// TIA Portal V17 export
// export: Created 2024-08-29T18:23:44.282771Z, ExportSetting WithDefaults, DisplayName Totally Integrated Automation Portal, DisplayVersion V17 Update 7, DisplayName TIA Portal Openness, DisplayVersion V17 Update 7, DisplayName TIA Portal Version Control Interface, DisplayVersion V17, DisplayName SINAMICS Startdrive Advanced, DisplayVersion V17 SP2, DisplayName SINAMICS Startdrive G110M, G120, G120C, G120D, G120P, G115D, DisplayVersion V17 SP2, DisplayName SINAMICS Startdrive G130, G150, S120, S150, SINAMICS MV, S210, DisplayVersion V17 SP2, DisplayName STEP 7 Professional, DisplayVersion V17 Update 7, DisplayName STEP 7 Safety, DisplayVersion V17 Update 6, DisplayName WinCC Advanced / Unified PC, DisplayVersion V17 Update 7
FUNCTION "modifyRecipe" : Void   // FC6, LAD
{ S7_Optimized_Access := 'TRUE' }
VERSION : 0.1
// stored: AutoNumber true, IsIECCheckEnabled false, SetENOAutomatically false, UDAEnableTagReadback false
   VAR_TEMP   // added for the SCL form of the ladder/FBD networks
      _w1 : Bool;
      _w2 : Bool;
   END_VAR
BEGIN

REGION Network 1: ERASE A STEP
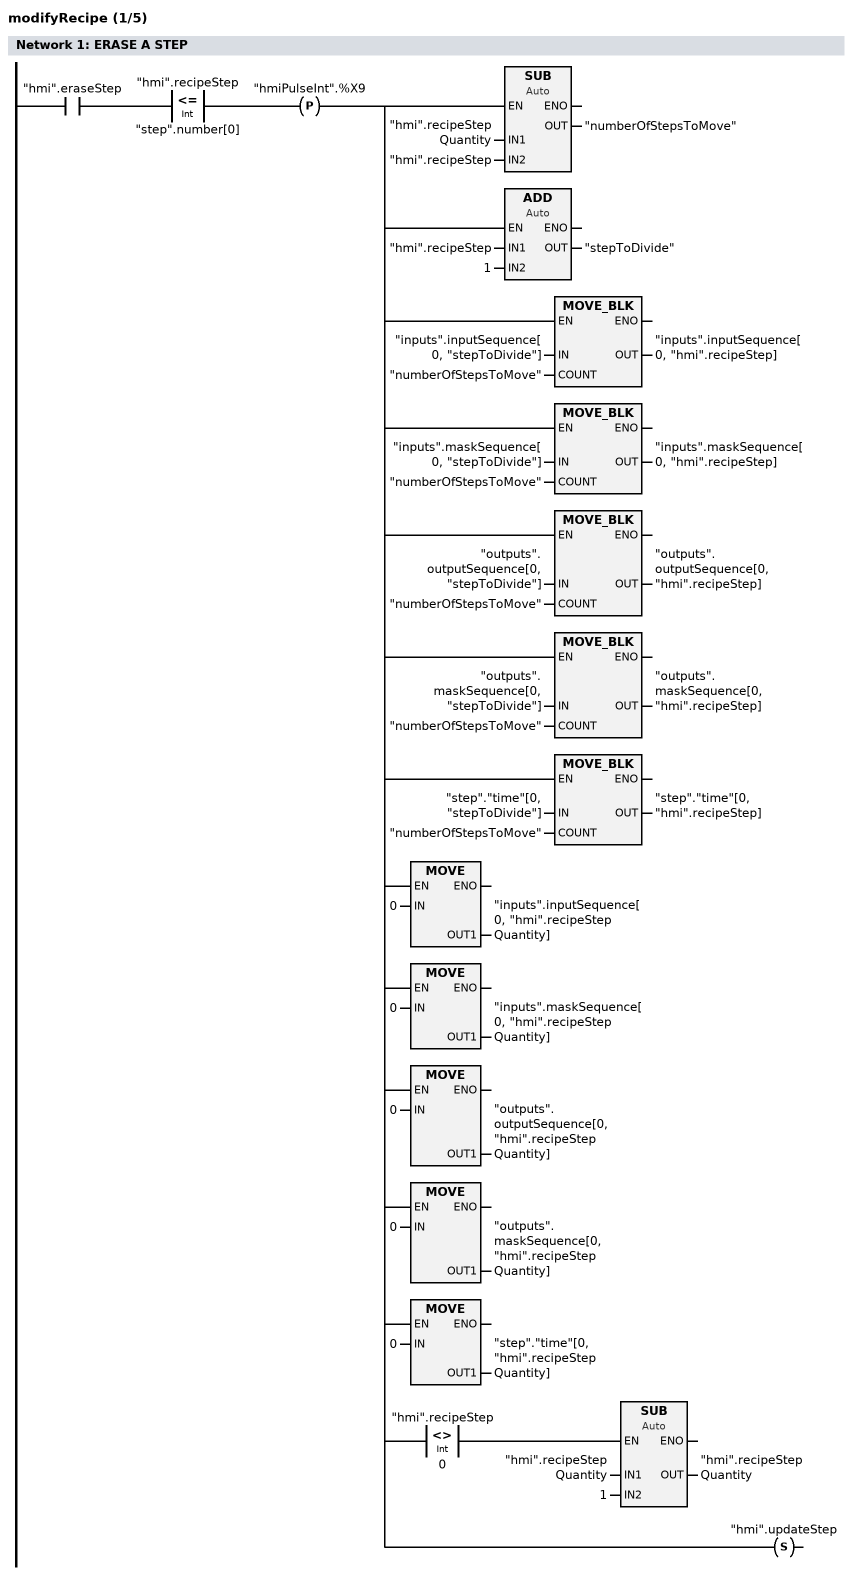
   #_w1 := "hmi".eraseStep AND ("hmi".recipeStep <= "step".number[0]);
   #_w2 := #_w1 AND NOT "hmiPulseInt".%X9;   // rising edge
   "hmiPulseInt".%X9 := #_w1;
   IF #_w2 THEN
       "numberOfStepsToMove" := "hmi".recipeStepQuantity - "hmi".recipeStep;
       "stepToDivide" := "hmi".recipeStep + 1;
       MOVE_BLK(IN := "inputs".inputSequence[0, "stepToDivide"],
                COUNT := "numberOfStepsToMove",
                OUT => "inputs".inputSequence[0, "hmi".recipeStep]);
       MOVE_BLK(IN := "inputs".maskSequence[0, "stepToDivide"],
                COUNT := "numberOfStepsToMove",
                OUT => "inputs".maskSequence[0, "hmi".recipeStep]);
       MOVE_BLK(IN := "outputs".outputSequence[0, "stepToDivide"],
                COUNT := "numberOfStepsToMove",
                OUT => "outputs".outputSequence[0, "hmi".recipeStep]);
       MOVE_BLK(IN := "outputs".maskSequence[0, "stepToDivide"],
                COUNT := "numberOfStepsToMove",
                OUT => "outputs".maskSequence[0, "hmi".recipeStep]);
       MOVE_BLK(IN := "step"."time"[0, "stepToDivide"],
                COUNT := "numberOfStepsToMove",
                OUT => "step"."time"[0, "hmi".recipeStep]);
       "inputs".inputSequence[0, "hmi".recipeStepQuantity] := 0;
       "inputs".maskSequence[0, "hmi".recipeStepQuantity] := 0;
       "outputs".outputSequence[0, "hmi".recipeStepQuantity] := 0;
       "outputs".maskSequence[0, "hmi".recipeStepQuantity] := 0;
       "step"."time"[0, "hmi".recipeStepQuantity] := 0;
   END_IF;
   IF #_w2 AND ("hmi".recipeStep <> 0) THEN "hmi".recipeStepQuantity := "hmi".recipeStepQuantity - 1; END_IF;
   IF #_w2 THEN "hmi".updateStep := TRUE; END_IF;
END_REGION

REGION Network 2: ADD A STEP
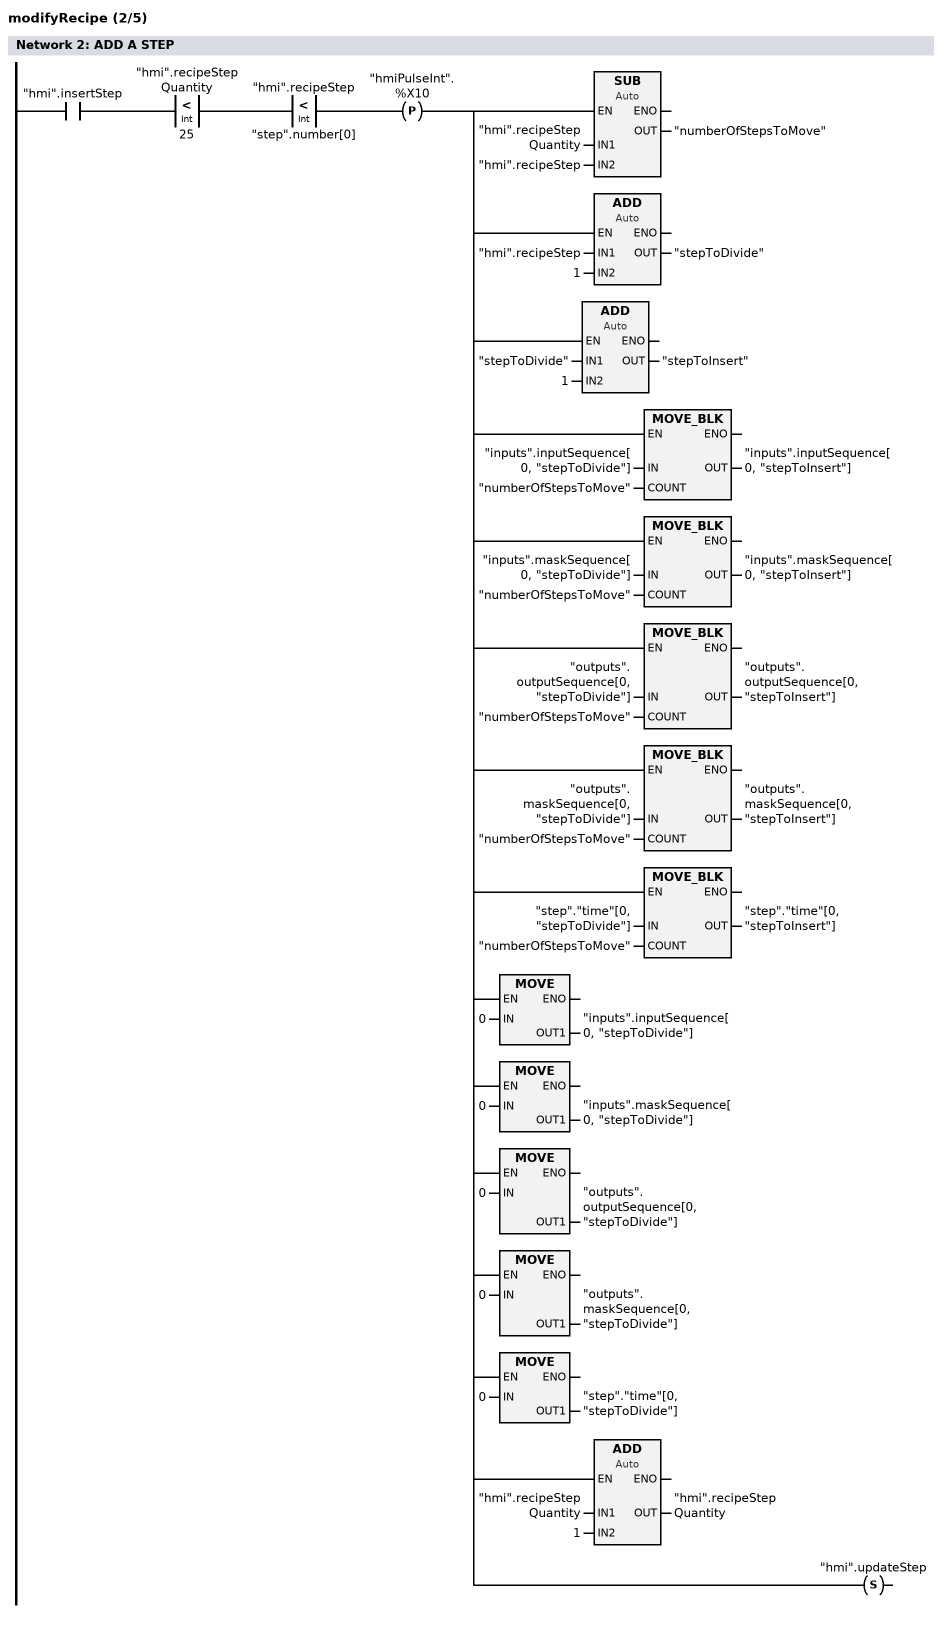
   #_w1 := "hmi".insertStep AND ("hmi".recipeStepQuantity < 25) AND ("hmi".recipeStep < "step".number[0]);
   #_w2 := #_w1 AND NOT "hmiPulseInt".%X10;   // rising edge
   "hmiPulseInt".%X10 := #_w1;
   IF #_w2 THEN
       "numberOfStepsToMove" := "hmi".recipeStepQuantity - "hmi".recipeStep;
       "stepToDivide" := "hmi".recipeStep + 1;
       "stepToInsert" := "stepToDivide" + 1;
       MOVE_BLK(IN := "inputs".inputSequence[0, "stepToDivide"],
                COUNT := "numberOfStepsToMove",
                OUT => "inputs".inputSequence[0, "stepToInsert"]);
       MOVE_BLK(IN := "inputs".maskSequence[0, "stepToDivide"],
                COUNT := "numberOfStepsToMove",
                OUT => "inputs".maskSequence[0, "stepToInsert"]);
       MOVE_BLK(IN := "outputs".outputSequence[0, "stepToDivide"],
                COUNT := "numberOfStepsToMove",
                OUT => "outputs".outputSequence[0, "stepToInsert"]);
       MOVE_BLK(IN := "outputs".maskSequence[0, "stepToDivide"],
                COUNT := "numberOfStepsToMove",
                OUT => "outputs".maskSequence[0, "stepToInsert"]);
       MOVE_BLK(IN := "step"."time"[0, "stepToDivide"],
                COUNT := "numberOfStepsToMove",
                OUT => "step"."time"[0, "stepToInsert"]);
       "inputs".inputSequence[0, "stepToDivide"] := 0;
       "inputs".maskSequence[0, "stepToDivide"] := 0;
       "outputs".outputSequence[0, "stepToDivide"] := 0;
       "outputs".maskSequence[0, "stepToDivide"] := 0;
       "step"."time"[0, "stepToDivide"] := 0;
       "hmi".recipeStepQuantity := "hmi".recipeStepQuantity + 1;
       "hmi".updateStep := TRUE;
   END_IF;
END_REGION

REGION Network 3: COPY A STEP
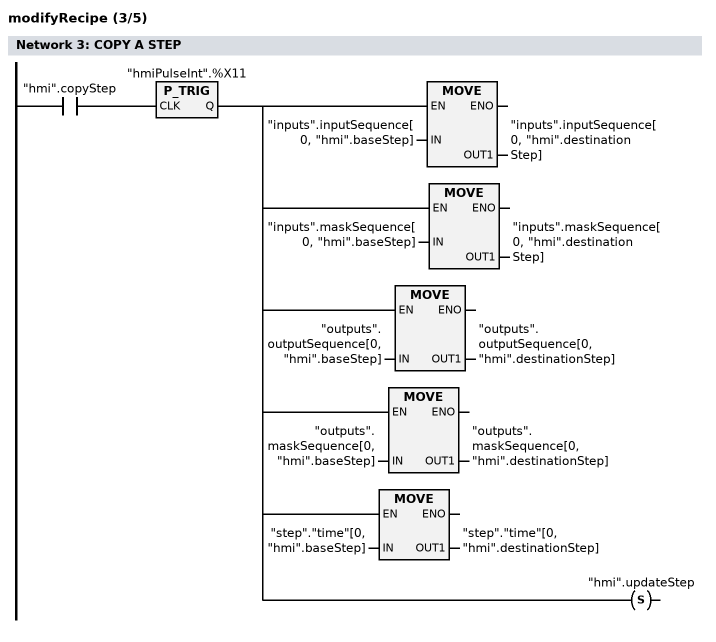
   RUNG wire#powerrail
      Contact( "hmi".copyStep )
      P_Trig( "hmiPulseInt".%X11 )
      wire#w1
      Move(in := "inputs".inputSequence[0, "hmi".baseStep], out1 => "inputs".inputSequence[0, "hmi".destinationStep])
   END_RUNG
   RUNG wire#w1
      Move(in := "inputs".maskSequence[0, "hmi".baseStep], out1 => "inputs".maskSequence[0, "hmi".destinationStep])
   END_RUNG
   RUNG wire#w1
      Move(in := "outputs".outputSequence[0, "hmi".baseStep], out1 => "outputs".outputSequence[0, "hmi".destinationStep])
   END_RUNG
   RUNG wire#w1
      Move(in := "outputs".maskSequence[0, "hmi".baseStep], out1 => "outputs".maskSequence[0, "hmi".destinationStep])
   END_RUNG
   RUNG wire#w1
      Move(in := "step"."time"[0, "hmi".baseStep], out1 => "step"."time"[0, "hmi".destinationStep])
   END_RUNG
   RUNG wire#w1
      S_Coil( "hmi".updateStep )
   END_RUNG
   // the same network as SCL:
   #_w1 := "hmi".copyStep AND NOT "hmiPulseInt".%X11;   // rising edge
   "hmiPulseInt".%X11 := "hmi".copyStep;
   IF #_w1 THEN
       "inputs".inputSequence[0, "hmi".destinationStep] := "inputs".inputSequence[0, "hmi".baseStep];
       "inputs".maskSequence[0, "hmi".destinationStep] := "inputs".maskSequence[0, "hmi".baseStep];
       "outputs".outputSequence[0, "hmi".destinationStep] := "outputs".outputSequence[0, "hmi".baseStep];
       "outputs".maskSequence[0, "hmi".destinationStep] := "outputs".maskSequence[0, "hmi".baseStep];
       "step"."time"[0, "hmi".destinationStep] := "step"."time"[0, "hmi".baseStep];
       "hmi".updateStep := TRUE;
   END_IF;
END_REGION

REGION Network 4: COPY SEQUENCE (COPY PART NUMBER)
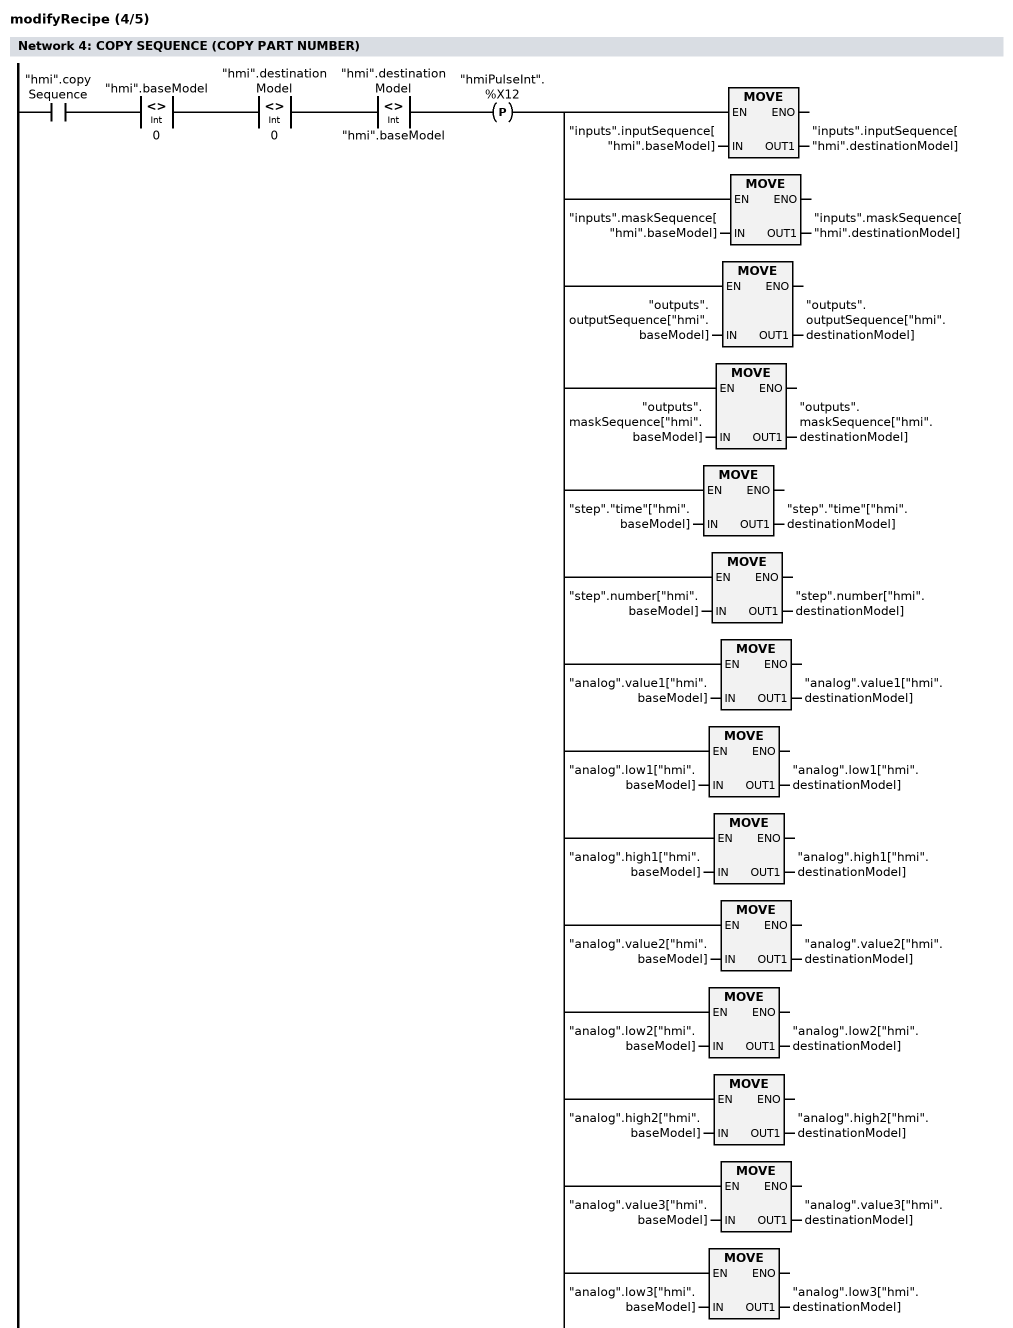
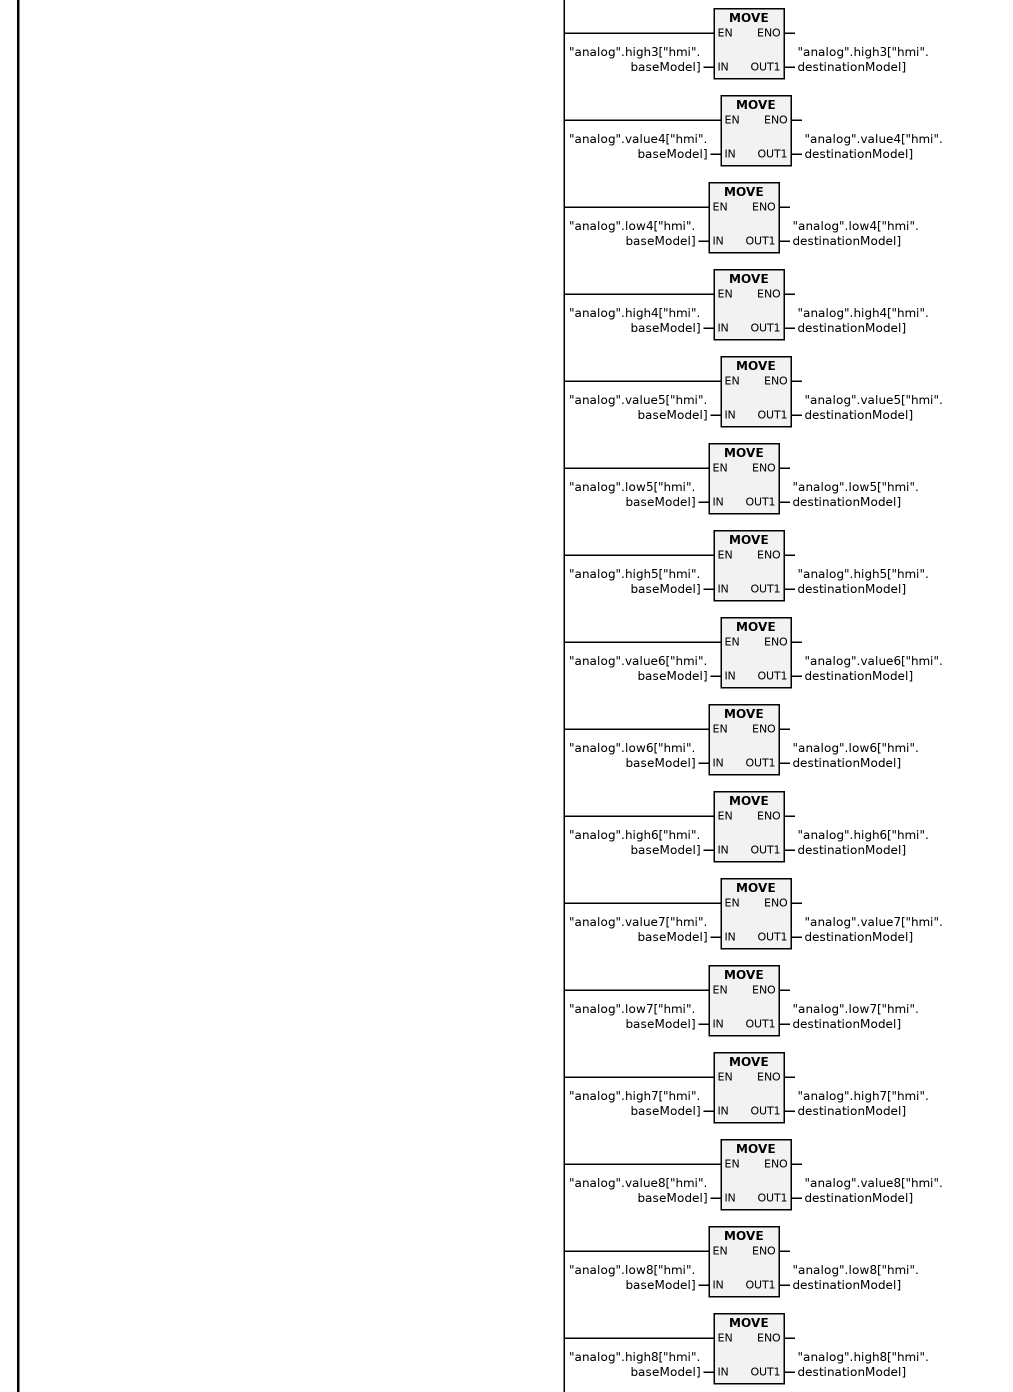
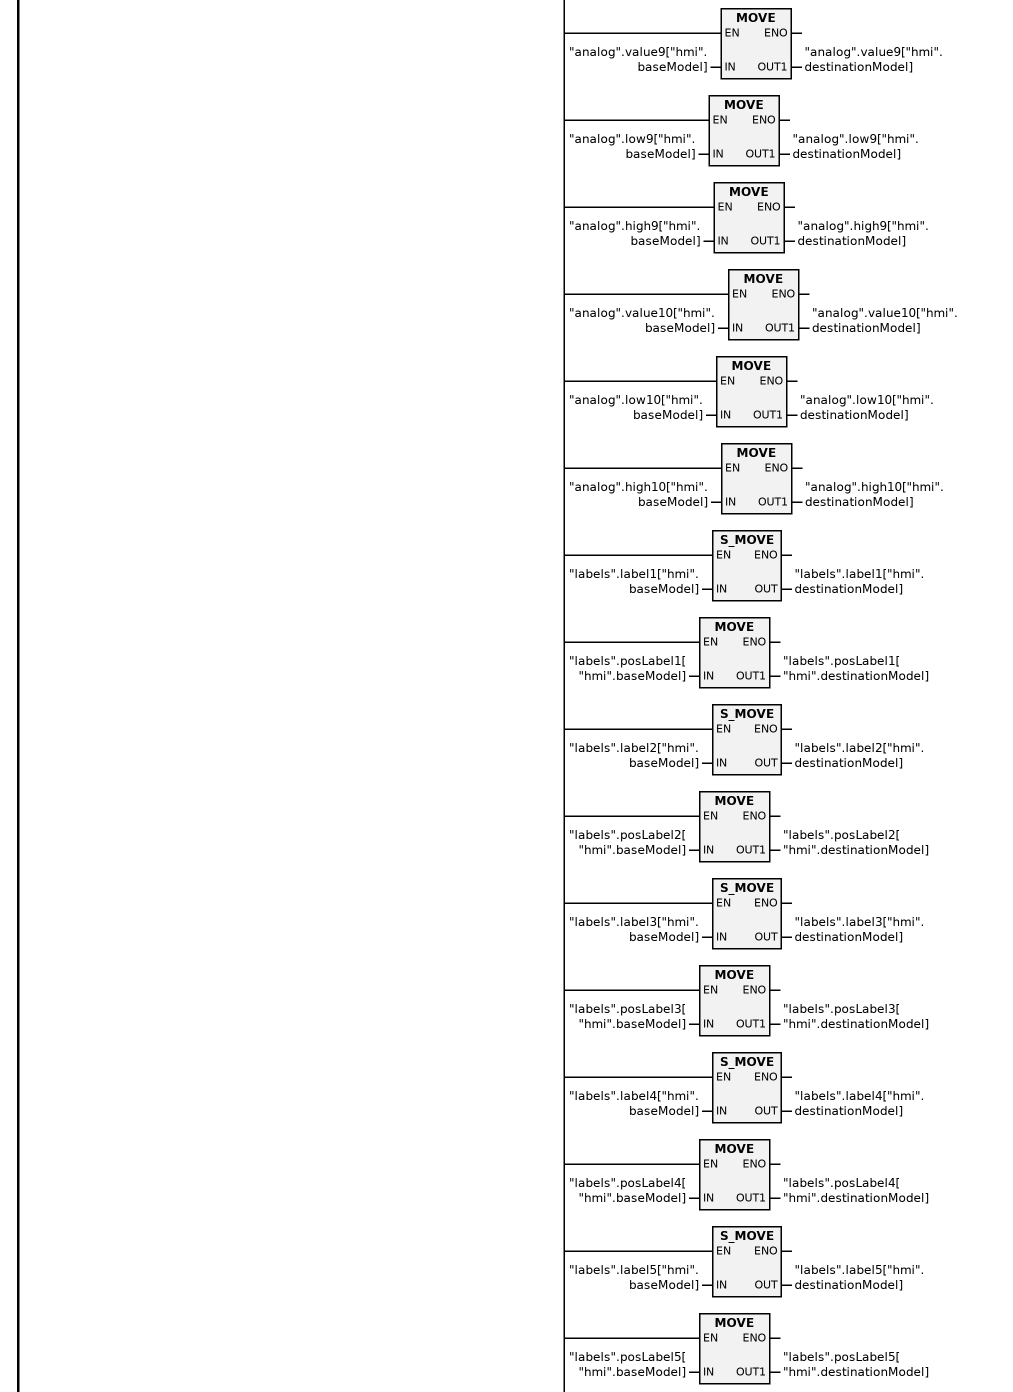
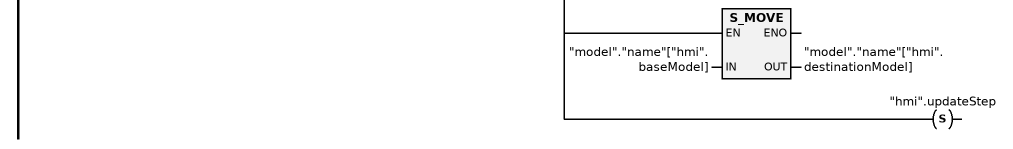
   RUNG wire#powerrail
      Contact( "hmi".copySequence )
      { S7_Templates := "SrcType := Int" } NE_Contact(in1 := "hmi".baseModel, in2 := 0)
      { S7_Templates := "SrcType := Int" } NE_Contact(in1 := "hmi".destinationModel, in2 := 0)
      { S7_Templates := "SrcType := Int" } NE_Contact(in1 := "hmi".destinationModel, in2 := "hmi".baseModel)
      P_Trig( "hmiPulseInt".%X12 )
      wire#w1
      Move(in := "inputs".inputSequence["hmi".baseModel], out1 => "inputs".inputSequence["hmi".destinationModel])
   END_RUNG
   RUNG wire#w1
      Move(in := "inputs".maskSequence["hmi".baseModel], out1 => "inputs".maskSequence["hmi".destinationModel])
   END_RUNG
   RUNG wire#w1
      Move(in := "outputs".outputSequence["hmi".baseModel], out1 => "outputs".outputSequence["hmi".destinationModel])
   END_RUNG
   RUNG wire#w1
      Move(in := "outputs".maskSequence["hmi".baseModel], out1 => "outputs".maskSequence["hmi".destinationModel])
   END_RUNG
   RUNG wire#w1
      Move(in := "step"."time"["hmi".baseModel], out1 => "step"."time"["hmi".destinationModel])
   END_RUNG
   RUNG wire#w1
      Move(in := "step".number["hmi".baseModel], out1 => "step".number["hmi".destinationModel])
   END_RUNG
   RUNG wire#w1
      Move(in := "analog".value1["hmi".baseModel], out1 => "analog".value1["hmi".destinationModel])
   END_RUNG
   RUNG wire#w1
      Move(in := "analog".low1["hmi".baseModel], out1 => "analog".low1["hmi".destinationModel])
   END_RUNG
   RUNG wire#w1
      Move(in := "analog".high1["hmi".baseModel], out1 => "analog".high1["hmi".destinationModel])
   END_RUNG
   RUNG wire#w1
      Move(in := "analog".value2["hmi".baseModel], out1 => "analog".value2["hmi".destinationModel])
   END_RUNG
   RUNG wire#w1
      Move(in := "analog".low2["hmi".baseModel], out1 => "analog".low2["hmi".destinationModel])
   END_RUNG
   RUNG wire#w1
      Move(in := "analog".high2["hmi".baseModel], out1 => "analog".high2["hmi".destinationModel])
   END_RUNG
   RUNG wire#w1
      Move(in := "analog".value3["hmi".baseModel], out1 => "analog".value3["hmi".destinationModel])
   END_RUNG
   RUNG wire#w1
      Move(in := "analog".low3["hmi".baseModel], out1 => "analog".low3["hmi".destinationModel])
   END_RUNG
   RUNG wire#w1
      Move(in := "analog".high3["hmi".baseModel], out1 => "analog".high3["hmi".destinationModel])
   END_RUNG
   RUNG wire#w1
      Move(in := "analog".value4["hmi".baseModel], out1 => "analog".value4["hmi".destinationModel])
   END_RUNG
   RUNG wire#w1
      Move(in := "analog".low4["hmi".baseModel], out1 => "analog".low4["hmi".destinationModel])
   END_RUNG
   RUNG wire#w1
      Move(in := "analog".high4["hmi".baseModel], out1 => "analog".high4["hmi".destinationModel])
   END_RUNG
   RUNG wire#w1
      Move(in := "analog".value5["hmi".baseModel], out1 => "analog".value5["hmi".destinationModel])
   END_RUNG
   RUNG wire#w1
      Move(in := "analog".low5["hmi".baseModel], out1 => "analog".low5["hmi".destinationModel])
   END_RUNG
   RUNG wire#w1
      Move(in := "analog".high5["hmi".baseModel], out1 => "analog".high5["hmi".destinationModel])
   END_RUNG
   RUNG wire#w1
      Move(in := "analog".value6["hmi".baseModel], out1 => "analog".value6["hmi".destinationModel])
   END_RUNG
   RUNG wire#w1
      Move(in := "analog".low6["hmi".baseModel], out1 => "analog".low6["hmi".destinationModel])
   END_RUNG
   RUNG wire#w1
      Move(in := "analog".high6["hmi".baseModel], out1 => "analog".high6["hmi".destinationModel])
   END_RUNG
   RUNG wire#w1
      Move(in := "analog".value7["hmi".baseModel], out1 => "analog".value7["hmi".destinationModel])
   END_RUNG
   RUNG wire#w1
      Move(in := "analog".low7["hmi".baseModel], out1 => "analog".low7["hmi".destinationModel])
   END_RUNG
   RUNG wire#w1
      Move(in := "analog".high7["hmi".baseModel], out1 => "analog".high7["hmi".destinationModel])
   END_RUNG
   RUNG wire#w1
      Move(in := "analog".value8["hmi".baseModel], out1 => "analog".value8["hmi".destinationModel])
   END_RUNG
   RUNG wire#w1
      Move(in := "analog".low8["hmi".baseModel], out1 => "analog".low8["hmi".destinationModel])
   END_RUNG
   RUNG wire#w1
      Move(in := "analog".high8["hmi".baseModel], out1 => "analog".high8["hmi".destinationModel])
   END_RUNG
   RUNG wire#w1
      Move(in := "analog".value9["hmi".baseModel], out1 => "analog".value9["hmi".destinationModel])
   END_RUNG
   RUNG wire#w1
      Move(in := "analog".low9["hmi".baseModel], out1 => "analog".low9["hmi".destinationModel])
   END_RUNG
   RUNG wire#w1
      Move(in := "analog".high9["hmi".baseModel], out1 => "analog".high9["hmi".destinationModel])
   END_RUNG
   RUNG wire#w1
      Move(in := "analog".value10["hmi".baseModel], out1 => "analog".value10["hmi".destinationModel])
   END_RUNG
   RUNG wire#w1
      Move(in := "analog".low10["hmi".baseModel], out1 => "analog".low10["hmi".destinationModel])
   END_RUNG
   RUNG wire#w1
      Move(in := "analog".high10["hmi".baseModel], out1 => "analog".high10["hmi".destinationModel])
   END_RUNG
   RUNG wire#w1
      S_Move(in := "labels".label1["hmi".baseModel], out => "labels".label1["hmi".destinationModel])
   END_RUNG
   RUNG wire#w1
      Move(in := "labels".posLabel1["hmi".baseModel], out1 => "labels".posLabel1["hmi".destinationModel])
   END_RUNG
   RUNG wire#w1
      S_Move(in := "labels".label2["hmi".baseModel], out => "labels".label2["hmi".destinationModel])
   END_RUNG
   RUNG wire#w1
      Move(in := "labels".posLabel2["hmi".baseModel], out1 => "labels".posLabel2["hmi".destinationModel])
   END_RUNG
   RUNG wire#w1
      S_Move(in := "labels".label3["hmi".baseModel], out => "labels".label3["hmi".destinationModel])
   END_RUNG
   RUNG wire#w1
      Move(in := "labels".posLabel3["hmi".baseModel], out1 => "labels".posLabel3["hmi".destinationModel])
   END_RUNG
   RUNG wire#w1
      S_Move(in := "labels".label4["hmi".baseModel], out => "labels".label4["hmi".destinationModel])
   END_RUNG
   RUNG wire#w1
      Move(in := "labels".posLabel4["hmi".baseModel], out1 => "labels".posLabel4["hmi".destinationModel])
   END_RUNG
   RUNG wire#w1
      S_Move(in := "labels".label5["hmi".baseModel], out => "labels".label5["hmi".destinationModel])
   END_RUNG
   RUNG wire#w1
      Move(in := "labels".posLabel5["hmi".baseModel], out1 => "labels".posLabel5["hmi".destinationModel])
   END_RUNG
   RUNG wire#w1
      S_Move(in := "model"."name"["hmi".baseModel], out => "model"."name"["hmi".destinationModel])
   END_RUNG
   RUNG wire#w1
      S_Coil( "hmi".updateStep )
   END_RUNG
   // the same network as SCL:
   #_w1 := "hmi".copySequence AND ("hmi".baseModel <> 0) AND ("hmi".destinationModel <> 0) AND ("hmi".destinationModel <> "hmi".baseModel);
   #_w2 := #_w1 AND NOT "hmiPulseInt".%X12;   // rising edge
   "hmiPulseInt".%X12 := #_w1;
   IF #_w2 THEN
       "inputs".inputSequence["hmi".destinationModel] := "inputs".inputSequence["hmi".baseModel];
       "inputs".maskSequence["hmi".destinationModel] := "inputs".maskSequence["hmi".baseModel];
       "outputs".outputSequence["hmi".destinationModel] := "outputs".outputSequence["hmi".baseModel];
       "outputs".maskSequence["hmi".destinationModel] := "outputs".maskSequence["hmi".baseModel];
       "step"."time"["hmi".destinationModel] := "step"."time"["hmi".baseModel];
       "step".number["hmi".destinationModel] := "step".number["hmi".baseModel];
       "analog".value1["hmi".destinationModel] := "analog".value1["hmi".baseModel];
       "analog".low1["hmi".destinationModel] := "analog".low1["hmi".baseModel];
       "analog".high1["hmi".destinationModel] := "analog".high1["hmi".baseModel];
       "analog".value2["hmi".destinationModel] := "analog".value2["hmi".baseModel];
       "analog".low2["hmi".destinationModel] := "analog".low2["hmi".baseModel];
       "analog".high2["hmi".destinationModel] := "analog".high2["hmi".baseModel];
       "analog".value3["hmi".destinationModel] := "analog".value3["hmi".baseModel];
       "analog".low3["hmi".destinationModel] := "analog".low3["hmi".baseModel];
       "analog".high3["hmi".destinationModel] := "analog".high3["hmi".baseModel];
       "analog".value4["hmi".destinationModel] := "analog".value4["hmi".baseModel];
       "analog".low4["hmi".destinationModel] := "analog".low4["hmi".baseModel];
       "analog".high4["hmi".destinationModel] := "analog".high4["hmi".baseModel];
       "analog".value5["hmi".destinationModel] := "analog".value5["hmi".baseModel];
       "analog".low5["hmi".destinationModel] := "analog".low5["hmi".baseModel];
       "analog".high5["hmi".destinationModel] := "analog".high5["hmi".baseModel];
       "analog".value6["hmi".destinationModel] := "analog".value6["hmi".baseModel];
       "analog".low6["hmi".destinationModel] := "analog".low6["hmi".baseModel];
       "analog".high6["hmi".destinationModel] := "analog".high6["hmi".baseModel];
       "analog".value7["hmi".destinationModel] := "analog".value7["hmi".baseModel];
       "analog".low7["hmi".destinationModel] := "analog".low7["hmi".baseModel];
       "analog".high7["hmi".destinationModel] := "analog".high7["hmi".baseModel];
       "analog".value8["hmi".destinationModel] := "analog".value8["hmi".baseModel];
       "analog".low8["hmi".destinationModel] := "analog".low8["hmi".baseModel];
       "analog".high8["hmi".destinationModel] := "analog".high8["hmi".baseModel];
       "analog".value9["hmi".destinationModel] := "analog".value9["hmi".baseModel];
       "analog".low9["hmi".destinationModel] := "analog".low9["hmi".baseModel];
       "analog".high9["hmi".destinationModel] := "analog".high9["hmi".baseModel];
       "analog".value10["hmi".destinationModel] := "analog".value10["hmi".baseModel];
       "analog".low10["hmi".destinationModel] := "analog".low10["hmi".baseModel];
       "analog".high10["hmi".destinationModel] := "analog".high10["hmi".baseModel];
       "labels".label1["hmi".destinationModel] := "labels".label1["hmi".baseModel];
       "labels".posLabel1["hmi".destinationModel] := "labels".posLabel1["hmi".baseModel];
       "labels".label2["hmi".destinationModel] := "labels".label2["hmi".baseModel];
       "labels".posLabel2["hmi".destinationModel] := "labels".posLabel2["hmi".baseModel];
       "labels".label3["hmi".destinationModel] := "labels".label3["hmi".baseModel];
       "labels".posLabel3["hmi".destinationModel] := "labels".posLabel3["hmi".baseModel];
       "labels".label4["hmi".destinationModel] := "labels".label4["hmi".baseModel];
       "labels".posLabel4["hmi".destinationModel] := "labels".posLabel4["hmi".baseModel];
       "labels".label5["hmi".destinationModel] := "labels".label5["hmi".baseModel];
       "labels".posLabel5["hmi".destinationModel] := "labels".posLabel5["hmi".baseModel];
       "model"."name"["hmi".destinationModel] := "model"."name"["hmi".baseModel];
       "hmi".updateStep := TRUE;
   END_IF;
END_REGION

REGION Network 5: COPY A STEP (#) FROM A PROGRAM (#) IN ANOTHER STEP (#) FROM ANOTHER PROGRAM (#)
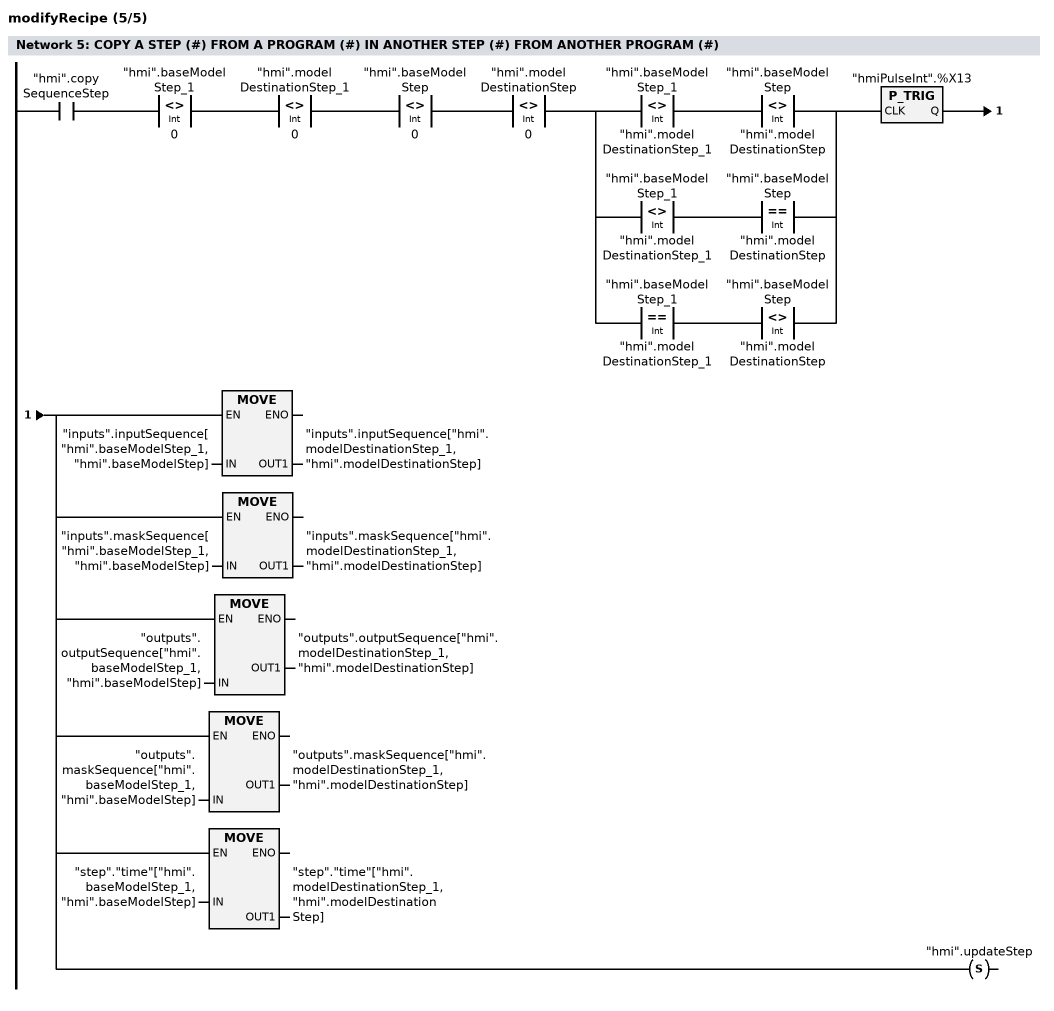
   RUNG wire#powerrail
      Contact( "hmi".copySequenceStep )
      { S7_Templates := "SrcType := Int" } NE_Contact(in1 := "hmi".baseModelStep_1, in2 := 0)
      { S7_Templates := "SrcType := Int" } NE_Contact(in1 := "hmi".modelDestinationStep_1, in2 := 0)
      { S7_Templates := "SrcType := Int" } NE_Contact(in1 := "hmi".baseModelStep, in2 := 0)
      { S7_Templates := "SrcType := Int" } NE_Contact(in1 := "hmi".modelDestinationStep, in2 := 0)
      wire#w1
      { S7_Templates := "SrcType := Int" } NE_Contact(in1 := "hmi".baseModelStep_1, in2 := "hmi".modelDestinationStep_1)
      { S7_Templates := "SrcType := Int" } NE_Contact(in1 := "hmi".baseModelStep, in2 := "hmi".modelDestinationStep)
      wire#w2
      P_Trig( "hmiPulseInt".%X13 )
      wire#w3
      Move(in := "inputs".inputSequence["hmi".baseModelStep_1, "hmi".baseModelStep], out1 => "inputs".inputSequence["hmi".modelDestinationStep_1, "hmi".modelDestinationStep])
   END_RUNG
   RUNG wire#w1
      { S7_Templates := "SrcType := Int" } NE_Contact(in1 := "hmi".baseModelStep_1, in2 := "hmi".modelDestinationStep_1)
      { S7_Templates := "SrcType := Int" } EQ_Contact(in1 := "hmi".baseModelStep, in2 := "hmi".modelDestinationStep)
   END_RUNG wire#w2
   RUNG wire#w1
      { S7_Templates := "SrcType := Int" } EQ_Contact(in1 := "hmi".baseModelStep_1, in2 := "hmi".modelDestinationStep_1)
      { S7_Templates := "SrcType := Int" } NE_Contact(in1 := "hmi".baseModelStep, in2 := "hmi".modelDestinationStep)
   END_RUNG wire#w2
   RUNG wire#w3
      Move(in := "inputs".maskSequence["hmi".baseModelStep_1, "hmi".baseModelStep], out1 => "inputs".maskSequence["hmi".modelDestinationStep_1, "hmi".modelDestinationStep])
   END_RUNG
   RUNG wire#w3
      Move(in := "outputs".outputSequence["hmi".baseModelStep_1, "hmi".baseModelStep], out1 => "outputs".outputSequence["hmi".modelDestinationStep_1, "hmi".modelDestinationStep])
   END_RUNG
   RUNG wire#w3
      Move(in := "outputs".maskSequence["hmi".baseModelStep_1, "hmi".baseModelStep], out1 => "outputs".maskSequence["hmi".modelDestinationStep_1, "hmi".modelDestinationStep])
   END_RUNG
   RUNG wire#w3
      Move(in := "step"."time"["hmi".baseModelStep_1, "hmi".baseModelStep], out1 => "step"."time"["hmi".modelDestinationStep_1, "hmi".modelDestinationStep])
   END_RUNG
   RUNG wire#w3
      S_Coil( "hmi".updateStep )
   END_RUNG
   // the same network as SCL:
   #_w1 := "hmi".copySequenceStep AND ("hmi".baseModelStep_1 <> 0) AND ("hmi".modelDestinationStep_1 <> 0) AND ("hmi".baseModelStep <> 0) AND ("hmi".modelDestinationStep <> 0) AND ((("hmi".baseModelStep_1 <> "hmi".modelDestinationStep_1) AND ("hmi".baseModelStep <> "hmi".modelDestinationStep)) OR (("hmi".baseModelStep_1 <> "hmi".modelDestinationStep_1) AND ("hmi".baseModelStep = "hmi".modelDestinationStep)) OR (("hmi".baseModelStep_1 = "hmi".modelDestinationStep_1) AND ("hmi".baseModelStep <> "hmi".modelDestinationStep)));
   #_w2 := #_w1 AND NOT "hmiPulseInt".%X13;   // rising edge
   "hmiPulseInt".%X13 := #_w1;
   IF #_w2 THEN
       "inputs".inputSequence["hmi".modelDestinationStep_1, "hmi".modelDestinationStep] := "inputs".inputSequence["hmi".baseModelStep_1, "hmi".baseModelStep];
       "inputs".maskSequence["hmi".modelDestinationStep_1, "hmi".modelDestinationStep] := "inputs".maskSequence["hmi".baseModelStep_1, "hmi".baseModelStep];
       "outputs".outputSequence["hmi".modelDestinationStep_1, "hmi".modelDestinationStep] := "outputs".outputSequence["hmi".baseModelStep_1, "hmi".baseModelStep];
       "outputs".maskSequence["hmi".modelDestinationStep_1, "hmi".modelDestinationStep] := "outputs".maskSequence["hmi".baseModelStep_1, "hmi".baseModelStep];
       "step"."time"["hmi".modelDestinationStep_1, "hmi".modelDestinationStep] := "step"."time"["hmi".baseModelStep_1, "hmi".baseModelStep];
       "hmi".updateStep := TRUE;
   END_IF;
END_REGION
END_FUNCTION
